FUNCTION_BLOCK FB_Tiger IMPLEMENTS I_AnimalTraits
VAR_INPUT
END_VAR
VAR_OUTPUT
END_VAR
VAR
END_VAR

{warning 'add method implementation '}
METHOD DietType : BOOL
END_METHOD

{warning 'add method implementation '}
METHOD IsDangerous : BOOL
END_METHOD

END_FUNCTION_BLOCK

(* stored: Version 1.1.0.1, ProductVersion 3.1.4024.16
   POU FB_Tiger: Id {7b4d2bb9-8e01-497f-8b2b-2c7fa30ab563}, SpecialFunc None
   Method DietType: Id {9bf16a33-2e09-4b3a-99a9-9ef9395ab37d}
   Method IsDangerous: Id {2eec1d60-d638-4634-a2f5-738303d2c1e8} *)
